// TIA Portal project "SQLStorage" (V15.1)

(* hardware
DEVICE "S71500/ET200MP station_1"  S7-1500 station
   slot 0: "Rail_0"  Rack  6ES7 590-1***0-0AA0
   slot 1: "PLC_1"  CPU 1511-1 PN  6ES7 511-1AK02-0AB0  V2.6
      slot 3: "CPU display_1"  6ES7591-1AA00-0AA0
DEVICE "PC station"  SIMATIC PC station
   slot 0: "PC station"  Rail  SIMATIC PC-Station  V1.0
      slot 125: "Stationmanager"  Station_Manager  V6.0.4
   slot 1: "IE general_1"  IE General  IE_CP  V8.2.0
   slot 3: "HMI_RT_1"  WinCC RT Advanced  6AV2 104-0xxxx-xxxx  15.1.0.0
      slot 33792: "Host interface"  Host interface
*)

// ===== PLC "PLC_1"  CPU 1511-1 PN =====

ORGANIZATION_BLOCK "Main"   // OB1, LAD, ProgramCycle
TITLE = "Main Program Sweep (Cycle)"
{ S7_Optimized_Access := 'TRUE' }
VERSION : 0.1
   VAR_INPUT
      Initial_Call : Bool;   // Initial call of this OB
      Remanence : Bool;   // =True, if remanent data are available
   END_VAR
BEGIN
END_ORGANIZATION_BLOCK

(* ===== HMI "HMI_RT_1" =====
system functions are stored by id; their names below are inferred from use

HMI tags "Default tag table"
   "HMI_Tag_1" : Int, internal
   "szDataBase" : WString[10], internal
   "szTableName" : WString[10], internal
   "szName_1" : WString[10], internal
   "szName_2" : WString[10], internal
   "szName_3" : WString[10], internal
   "nDat_No" : Int, internal
   "nValue_1" : WString[10], internal
   "nValue_2" : Int, internal
   "nValue_3" : Int, internal

screen "databaseManagement" 640x480
   TextField "Text field_1" at 264,101 size 122x22; Text 'Database Name'
   IOField "I/O field_1" at 255,139 size 139x32; FormatPattern ???????????????
      ProcessValue <- "szDataBase"
   Button "Button_1" at 180,196 size 96x43; TextOff 'Add DB'
      on Press: "createDB"()
   Button "Button_2" at 373,196 size 96x43; TextOff 'Remove DB'
      on Press: "deleteDB"()
   Button "Button_3" at 37,376 size 96x32; TextOff 'Traceback'
      on Press: function_ef3f5d25("Alarm window_1", -1)
   Button "Button_4" at 465,376 size 139x32; TextOff 'Storage Control'
      on Press: ActivateScreen("storageControl", 0)

screen "storageControl" 640x480
   TextField "Text field_1" at 241,134 size 163x22; Text 'Storage Management'
   Button "Button_1" at 200,164 size 245x32; TextOff 'Create DB / Delete DB'
      on Press: ActivateScreen("databaseManagement", 0)
   Button "Button_2" at 200,203 size 245x32; TextOff 'Create Table'
      on Press: ActivateScreen("createTable", 0)
   Button "Button_3" at 200,244 size 245x32; TextOff 'Delete Table'
      on Press: ActivateScreen("deleteTable", 0)
   Button "Button_4" at 200,284 size 245x32; TextOff 'Add Data'
      on Press: ActivateScreen("addData", 0)

screen "createTable" 640x480
   TextField "Text field_1" at 259,39 size 122x22; Text 'Database Name'
   IOField "I/O field_1" at 257,76 size 125x32; FormatPattern ??????????
      ProcessValue <- "szDataBase"
   TextField "Text field_2" at 273,124 size 93x22; Text 'Table Name'
   IOField "I/O field_2" at 257,161 size 125x32; FormatPattern ??????????
      ProcessValue <- "szTableName"
   TextField "Text field_3" at 115,232 size 74x22; Text 'Column 1'
   TextField "Text field_4" at 115,277 size 74x22; Text 'Column 2'
   TextField "Text field_5" at 115,325 size 74x22; Text 'Column 3'
   IOField "I/O field_3" at 257,232 size 125x32; FormatPattern ??????????
      ProcessValue <- "szName_1"
   IOField "I/O field_4" at 257,277 size 125x32; FormatPattern ??????????
      ProcessValue <- "szName_2"
   IOField "I/O field_5" at 257,325 size 125x32; FormatPattern ??????????
      ProcessValue <- "szName_3"
   Button "Button_1" at 481,421 size 138x32; TextOff 'Storage Control'
      on Press: ActivateScreen("storageControl", 0)
   Button "Button_2" at 257,395 size 124x39; TextOff 'Create Table'
      on Press: "createTable"()

screen "deleteTable" 640x480
   TextField "Text field_1" at 259,113 size 122x22; Text 'Database Name'
   IOField "I/O field_1" at 258,150 size 125x32; FormatPattern ??????????
      ProcessValue <- "szDataBase"
   TextField "Text field_2" at 274,198 size 93x22; Text 'Table Name'
   IOField "I/O field_2" at 258,235 size 125x32; FormatPattern ??????????
      ProcessValue <- "szTableName"
   Button "Button_1" at 481,421 size 138x32; TextOff 'Storage Control'
      on Press: ActivateScreen("storageControl", 0)
   Button "Button_2" at 259,304 size 124x39; TextOff 'Delete Table'
      on Press: "deleteTable"()

screen "addData" 640x480
   TextField "Text field_1" at 259,29 size 122x22; Text 'Database Name'
   IOField "I/O field_1" at 257,66 size 125x32; FormatPattern ??????????
      ProcessValue <- "szDataBase"
   TextField "Text field_2" at 273,114 size 93x22; Text 'Table Name'
   IOField "I/O field_2" at 257,151 size 125x32; FormatPattern ??????????
      ProcessValue <- "szTableName"
   TextField "Text field_3" at 58,262 size 61x22; Text 'Value 1'
   TextField "Text field_4" at 58,307 size 61x22; Text 'Value 2'
   TextField "Text field_5" at 58,355 size 61x22; Text 'Value 3'
   IOField "I/O field_3" at 200,262 size 236x32; FormatPattern ??????????
      ProcessValue <- "nValue_1"
   IOField "I/O field_4" at 200,307 size 237x32; FormatPattern s99999
      ProcessValue <- "nValue_2"
   IOField "I/O field_5" at 200,355 size 237x32; FormatPattern s99999
      ProcessValue <- "nValue_3"
   Button "Button_1" at 473,420 size 138x32; TextOff 'Storage Control'
      on Press: ActivateScreen("storageControl", 0)
   Button "Button_2" at 280,403 size 92x28; TextOff 'Add Data'
      on Press: "addData"()
   TextField "Text field_6" at 57,213 size 62x22; Text 'Dat_No'
   IOField "I/O field_6" at 199,213 size 237x32; FormatPattern s99999
      ProcessValue <- "nDat_No"

VB script "createDB"
   Dim connection, result, db_data
   On Error Resume Next
   
   Set connection = CreateObject("ADODB.Connection") 'database connection
   Set result = CreateObject("ADODB.Recordset") 'connection result
   
   connection.open = "Provider=MSDASQL; DSN=Database_1"
   
   If Err.Number <> 0 Then
   	bfde4b54-0db7-4817-8032-87127bf19bb9 "Error #" & Err.Number & " " & Err.Description
   	Err.Clear
   	Exit Sub
   End If
   
   db_data = "CREATE DATABASE " &  SmartTags("szDataBase")
   Set result = connection.Execute(db_data)
   
   If Err.Number <> 0 Then
   	bfde4b54-0db7-4817-8032-87127bf19bb9 "Error #" & Err.Number & " " & Err.Description
   	Err.Clear
   	Exit Sub
   End If
   
   connection.close
   Set connection = Nothing
   Set result = Nothing

VB script "deleteDB"
   Dim connection, result, db_data
   On Error Resume Next
   
   Set connection = CreateObject("ADODB.Connection") 'database connection
   Set result = CreateObject("ADODB.Recordset") 'connection result
   
   connection.open = "Provider=MSDASQL; DSN=Database_1"
   
   If Err.Number <> 0 Then
   	bfde4b54-0db7-4817-8032-87127bf19bb9 "Error #" & Err.Number & " " & Err.Description
   	Err.Clear
   	Exit Sub
   End If
   
   db_data = "DROP DATABASE " &  SmartTags("szDataBase")
   Set result = connection.Execute(db_data)
   
   If Err.Number <> 0 Then
   	bfde4b54-0db7-4817-8032-87127bf19bb9 "Error #" & Err.Number & " " & Err.Description
   	Err.Clear
   	Exit Sub
   End If
   
   connection.close
   Set connection = Nothing
   Set result = Nothing

VB script "createTable"
   Dim connection, result, db_data
   On Error Resume Next
   
   Set connection = CreateObject("ADODB.Connection") 'database connection
   Set result = CreateObject("ADODB.Recordset") 'connection result
   
   connection.open = "Provider=MSDASQL; Initial Catalog=" & SmartTags("szDataBase") & _
   				  ";DSN=Database_1"
   
   If Err.Number <> 0 Then
   	bfde4b54-0db7-4817-8032-87127bf19bb9 "Error #" & Err.Number & " " & Err.Description
   	Err.Clear
   	Exit Sub
   End If
   
   db_data = "CREATE TABLE " & SmartTags("szTableName") & " (Nr SMALLINT, " _
   		  & SmartTags("szName_1") & " CHAR(30), " & SmartTags("szName_2") & " SMALLINT, " _
   		  & SmartTags("szName_3") & " SMALLINT)" 
   
   Set result = connection.Execute(db_data)
   
   If Err.Number <> 0 Then
   	bfde4b54-0db7-4817-8032-87127bf19bb9 "Error #" & Err.Number & " " & Err.Description
   	Err.Clear
   	Exit Sub
   End If
   
   connection.close
   Set connection = Nothing
   Set result = Nothing

VB script "deleteTable"
   Dim connection, result, db_data
   On Error Resume Next
   
   Set connection = CreateObject("ADODB.Connection") 'database connection
   Set result = CreateObject("ADODB.Recordset") 'connection result
   
   connection.open = "Provider=MSDASQL; Initial Catalog=" & SmartTags("szDataBase") & _
   				  ";DSN=Database_1"
   
   If Err.Number <> 0 Then
   	bfde4b54-0db7-4817-8032-87127bf19bb9 "Error #" & Err.Number & " " & Err.Description
   	Err.Clear
   	Exit Sub
   End If
   
   db_data = "DROP TABLE " & SmartTags("szTableName") 
   
   Set result = connection.Execute(db_data)
   
   If Err.Number <> 0 Then
   	bfde4b54-0db7-4817-8032-87127bf19bb9 "Error #" & Err.Number & " " & Err.Description
   	Err.Clear
   	Exit Sub
   End If
   
   connection.close
   Set connection = Nothing
   Set result = Nothing

VB script "addData"
   Dim connection, result, db_data
   On Error Resume Next
   
   Set connection = CreateObject("ADODB.Connection") 'database connection
   Set result = CreateObject("ADODB.Recordset") 'connection result
   
   connection.open = "Provider=MSDASQL; Initial Catalog=" & SmartTags("szDataBase") & _
   				  ";DSN=Database_1"
   
   If Err.Number <> 0 Then
   	bfde4b54-0db7-4817-8032-87127bf19bb9 "Error #" & Err.Number & " " & Err.Description
   	Err.Clear
   	Exit Sub
   End If
   
   db_data = "SELECT * FROM " & SmartTags("szTableName") & " WHERE Nr = " & SmartTags("nDat_No") '* = all data
   
   Set result = connection.Execute(db_data)
   
   If Err.Number <> 0 Then
   	bfde4b54-0db7-4817-8032-87127bf19bb9 "Error #" & Err.Number & " " & Err.Description
   	Err.Clear
   	Exit Sub
   End If
   
   If Not (result.EOF And result.BOF) Then
   	bfde4b54-0db7-4817-8032-87127bf19bb9 "Dat No. exists already!"
   	result.close
   Else
   	db_data = "INSERT INTO " & SmartTags("szTableName") & " VALUES ('" & SmartTags("nDat_No") & _
   			  "','" & SmartTags("nValue_1") & "' , '" & SmartTags("nValue_2") &_
   			  "','" & SmartTags("nValue_3") & "')"
   	
   	Set result = connection.Execute(db_data)
   End If
   
   connection.close
   Set connection = Nothing
   Set result = Nothing
*)